INTERFACE I_SnappySetupConfigBuild

METHOD Build : HRESULT
VAR_INPUT
END_VAR
END_METHOD

END_INTERFACE

(* stored: Version 1.1.0.1, ProductVersion 3.1.4026.18
   Itf I_SnappySetupConfigBuild: Id {54ff1816-587c-4adf-8108-05ae72a52104}
   Method Build: Id {3eefaa5b-d67b-489f-9887-46326278cddd} *)
